// TIA Portal V16 export
// export: Created 2023-03-29T11:05:02.9769249Z, ExportSetting WithDefaults, DisplayName Totally Integrated Automation Portal, DisplayVersion V16 Update 6, DisplayName TIA Portal Version Control Interface, DisplayVersion V16 Update 2, DisplayName TIA Portal Openness, DisplayVersion V16 Update 6, DisplayName STEP 7 Professional, DisplayVersion V16 Update 6, DisplayName STEP 7 Safety, DisplayVersion V16, DisplayName WinCC Advanced, DisplayVersion V16 Update 6
DATA_BLOCK "dbtags_Sterowanie"   // DB1
{ S7_Optimized_Access := 'FALSE' }
VERSION : 0.1
// stored: AutoNumber false, DBAccessibleFromOPCUA true, IsOnlyStoredInLoadMemory false, IsWriteProtectedInAS false
   VAR RETAIN
      PID_Compact : Struct
         Setpoint : Real := 1.5;
         Input : Real;
         Input_PER : Int;
         Disturbance : Real;
         ManualEnable : Bool;
         ManualValue : Real;
         ErrorAck : Bool;
         Reset : Bool;
         ModeActivate : Bool;
         Mode : Int := 3;
         ScaledInput : Real;
         Output : Real;
         Output_PER : Int;
         Output_PWM : Bool;
         SetpointLimit_H : Bool;
         SetpointLimit_L : Bool;
         InputWarning_H : Bool;
         InputWarning_L : Bool;
         State : Int;
         Error : Bool;
         ErrorBits : DWord;
      END_STRUCT;
      Tuning : Struct
         Mode : Int := 1;
         Mode_visible : Bool;
         SUT_visible : Bool;
         TIR_visible : Bool;
         last_state : Int;
      END_STRUCT;
      HMI : Struct
         PhysicalUnit : String[5] := '1/min';
         Output_PWM_USInt : USInt;
         "position reached" : Bool;
         ManualMode_visible : Bool;
         Setpoint_limited : Bool;
         ErrorBits_Int : Int;
         ErrorAck_Int : Int;
         Warning_Int : Int;
         ErrorAck_Int_edge : Bool;   // pamięć zbocza reset PID po error
         ErrorAck : Bool;   // reset błędu PID
         Acknowledge_visible : Bool;
      END_STRUCT;
      Speed : Struct
         encoder : Real;
         rpm : Real;
      END_STRUCT;
      SetupControlPompownia : Struct
         SV : Real := 2.0;
         r_Pv_Norm_OUT_2 : Real := 10.0;   // Zakres górny wejścia In_PER_PID
         r_Pv_Norm_OUT_1 : Real := 0.0;   // Zakres dolny wejścia In_PER_PID
         r_Lmn_Hlm : Real := 100.0;   // Ograniczenie górne wartości procesowej [%] MV
         r_Lmn_Llm : Real := 0.0;   // Ograniczenie dolne wartości procesowej [%] MV
         r_Sp_Hlm : Real := 10.0;   // Ograniczenie H zakresu zadawania wartości ciśnienie SV
         r_Sp_Llm : Real := 0.0;   // Ograniczenie L zakresu zadawania wartości ciśnienia SV
         r_Pv_HWrn : Real;   // Ostrzeżenie wysoki dla PV
         r_Pv_LWrn : Real;   // Ostrzeżenie niski dla PV
         r_Pv_Hlm : Real := 16.0;   // Przetwornik Limit górny
         r_Pv_Llm : Real := 0.0;   // Przetwornik Limit dlolny
         Time_ONK1 : Int := 20;
         Time_ONK2 : Int := 60;
         Time_OFFK1 : Int := 15;
         Time_OFFK2 : Int := 5;
         TimeHz : Int := 10;
         NO4_Cureent : Real;   // Aktualna zawartość amoniaku
         CureentValue_O2_1 : Real;   // Przyrost ciśnienia 1
         CureentValue_O2_2 : Real;   // Przyrost ciścienia 2
         Data_sek1 : Int;   // Licznik sekund dla pomiaru nr1 funkcji Calculation_of_the_increment
         Data_sek2 : Int;   // Licznik sekund dla pomiaru nr2 funkcji Calculation_of_the_increment
         Static_1 : Word;
         Z11_Status : Word;   // Status napędu copia z SCADA
         Z12_Status : Word;   // Status napędu copia z SCADA
         Static_2 : Real;
         Switch_Aut_Rem_Pompy : Bool;   // Bit przełacznika trybu pracy pomp
         tagsdbSwitch_ModelSterowania : Word;   // Wybur model sterowania0- wyłączone, 1- Dosilanie, 2- Przetłączanie, 3- Automat, 4- Ręczne
         barMax_Manual_Hz : Real := 5.0;   // Instancja wartości zadawanej w trybie manual do regulatora PID gdy ciśnienie w rurociągu max
         CurrentMax_Manual_Hz : Real := 5.0;   // Instancja wartości zadawanej w trybie manual do regulatora PID gdy przeciążony falownik
         Statut_Motor : Byte;   // Byte stanu gotowości pomp
         Mem_Res_setCMD_MC_P1 : Bool;   // Znacznik 50 Hz podtrzymanie przełączenia na sieć
         Mem_Res_setCMD_MC_P2 : Bool;   // Znacznik 50 Hz podtrzymanie przełączenia na sieć
         Mem_Res_setCMD_MC_P3 : Bool;   // Znacznik 50 Hz podtrzymanie przełączenia na sieć
         Switch_In_Analog_Mudbas : Bool;   // Bit przełączeania pomiędzy sygnałem bar z wej analog / Modbus
         PV_HWrn_correction : Real;   // Wspóczninik służący wprowadzeniu korekty ostrzeżenia przekroczenia wartości zadanej ciśnienie
         PV_LWrn_correction : Real;   // Wspóczninik służący wprowadzeniu korekty ostrzeżenia zbyt niskia wartości ciśnieniea w stosunku do zadanej
         TimerSet_O2_Up : IEC_TIMER;   // Czas opóżninia podniesienia zadanej wartości ciśnienia
         TimerSet_O2_Down : IEC_TIMER;   // Czas opóżninia obniżenia zadanej wartości ciśnienia
         Pv_Llm_B8 : Real := -1.0;   // Limit dolny przetwornika ciśnienie B8
         Pv_Hlm_B8 : Real := 2.0;   // Limit górny przetwornika ciśnienia B8
         set_a : Int;
         set_b : Int := 0;
         Setpoint_Inverter_Pompy { ExternalAccessible := 'False'; ExternalVisible := 'False'; ExternalWritable := 'False'} : Real;   // Wartość zadana Hz odczytane z Modbus
         Frequency_inverter_Pompy { ExternalAccessible := 'False'; ExternalVisible := 'False'; ExternalWritable := 'False'} : Real;   // Aktualne Hz silniku odczytane z Modbus
         MotorCurrent_Inverter_Pompy { ExternalAccessible := 'False'; ExternalVisible := 'False'; ExternalWritable := 'False'} : Real;   // Prąd na silniku zasilanym z falownika odczytane z Modbus
         NormalCurrent_InverterPompy { ExternalAccessible := 'False'; ExternalVisible := 'False'; ExternalWritable := 'False'} : Real;   // Prąd nominalny falownika odczytane z Modbus
         MaxCurrent_Inverter_Pompy { ExternalAccessible := 'False'; ExternalVisible := 'False'; ExternalWritable := 'False'} : Real;   // Prad Max krótkotrwały odczytane z Modbus
         OverTemp_InverterPompy { ExternalAccessible := 'False'; ExternalVisible := 'False'; ExternalWritable := 'False'} : Word;
         OverVolta_InverterPompy { ExternalAccessible := 'False'; ExternalVisible := 'False'; ExternalWritable := 'False'} : Word;
         PIF_Reset : IEC_TIMER;   // impuls resetu regulatora PID 1
         mbAdresMPP04_Q1 : Word := 6;   // Adres modbus przepływomierz pompownia
         mbAdresPompy : Word := 26;   // Adres modbus falownik
         mbAdresMPP04_Q2 : Word;   // Adres modbus przepływomierz magistrala - w Stacji Zasuw
         mbAdres_IDslave : Word := 2;   // Adres modbus MT101
         SubPV_K1 : Real := 0.6;   // Wspólczynnik pomniejszenia wyliczanego ciśnienia napotrzeby wyłączenia dodatowej pompy
         SubPV_K2 : Real := 0.45;   // Wspólczynnik pomniejszenia wyliczanego ciśnieia napotrzeby wyłączenia dodatowej pompy
         Setpoint_Inverter_a { ExternalAccessible := 'False'; ExternalVisible := 'False'; ExternalWritable := 'False'} : Real;   // Wartość zadana Hz odczytane z Modbus
         Frequency_inverter_a { ExternalAccessible := 'False'; ExternalVisible := 'False'; ExternalWritable := 'False'} : Real;   // Aktualne Hz silniku odczytane z Modbus
         MotorCurrent_Inverter_a { ExternalAccessible := 'False'; ExternalVisible := 'False'; ExternalWritable := 'False'} : Real;   // Prąd na silniku zasilanym z falownika odczytane z Modbus
         NormalCurrent_Inverter_a { ExternalAccessible := 'False'; ExternalVisible := 'False'; ExternalWritable := 'False'} : Real;   // Prąd nominalny falownika odczytane z Modbus
         MaxCurrent_Inverter_a { ExternalAccessible := 'False'; ExternalVisible := 'False'; ExternalWritable := 'False'} : Real;   // Prad Max krótkotrwały odczytane z Modbus
         OverTemp_InverterPomp { ExternalAccessible := 'False'; ExternalVisible := 'False'; ExternalWritable := 'False'} : Word;
         OverVolta_InverterPomp { ExternalAccessible := 'False'; ExternalVisible := 'False'; ExternalWritable := 'False'} : Word;
         set_barDN500_B5 { ExternalAccessible := 'False'; ExternalVisible := 'False'; ExternalWritable := 'False'} : Real;   // Zadane ciśnienie dosilanie DN500 na czujniku B5
         set_barDN225_B6 { ExternalAccessible := 'False'; ExternalVisible := 'False'; ExternalWritable := 'False'} : Real;   // Zadane ciśnienie przetłacania DN225 na czujniku B6
         MotorCurrent_Inverter_b { ExternalAccessible := 'False'; ExternalVisible := 'False'; ExternalWritable := 'False'} : Real;   // Prąd na silniku zasilanym z falownika odczytane z Modbus
         NormalCurrent_Inverter_b { ExternalAccessible := 'False'; ExternalVisible := 'False'; ExternalWritable := 'False'} : Real;   // Prąd nominalny falownika odczytane z Modbus
         MaxCurrent_Inverter_b { ExternalAccessible := 'False'; ExternalVisible := 'False'; ExternalWritable := 'False'} : Real;   // Prad Max krótkotrwały odczytane z Modbus
         OverTemp_Inverter_b { ExternalAccessible := 'False'; ExternalVisible := 'False'; ExternalWritable := 'False'} : Word;
         OverVolta_Inverter_b { ExternalAccessible := 'False'; ExternalVisible := 'False'; ExternalWritable := 'False'} : Word;
         actOverCurrent_set : Real;   // Zakres ograniczenia prądowego.
         actOverCurrent_set_a : Real := 0.0;   // Zakres ograniczenia prądowego.
         actOverCurrent_set_b : Real := 0.0;   // Zakres ograniczenia prądowego.
         AnalogFrequency_inverter_a { ExternalAccessible := 'False'; ExternalVisible := 'False'; ExternalWritable := 'False'} : Real;   // Aktualne Hz silniku odczytane z Analog
         AnalogFrequency_inverter_b { ExternalAccessible := 'False'; ExternalVisible := 'False'; ExternalWritable := 'False'} : Real := 0.0;   // Aktualne Hz silniku odczytane z Analog
         MaxHour_InverterBlowerWork : Word := 43200;   // Maksymalny czas pracy pracy ciągłej na falowniku dla kompresorów 43200sek = 12h
         TimerSet_Hz_Up_a : IEC_TIMER;
         TimerSet_Hz_Down_a : IEC_TIMER;
         TimerSet_Hz_Up_b : IEC_TIMER;
         TimerSet_Hz_Down_b : IEC_TIMER;
         TimerGen_Hz_Up_a : IEC_TIMER;
         TimerGen_Hz_Down_a : IEC_TIMER;
         TimerGen_Hz_Up_b : IEC_TIMER;
         TimerGen_Hz_Down_b : IEC_TIMER;
         Mem_Res_setCMD_MC_P4 : Bool;   // Znacznik 50 Hz podtrzymanie przełączenia na sieć
         "MPP04_1Master.mode" : Byte := 0;
         "MPP04_2Master.mode" : Byte := 0;
         "Fal_2Master.mode_1" : Byte := 0;
         "Slave_2Master.mode_2" : Byte := 2;
      END_STRUCT;
      "Paramaetry _Zbiorniki" : Struct   // parametry sterowania
         set_poziom_napełniania : Real := 550.0;   // wartość zadana poziomu napełniania
         set_poziom_opróżniania : Real := 30.0;   // wartość zadana poziomu opróżniania
         set_bity_sterowania_napęami_1 : Word;   // bity sterowania napędami
         set_bity_sterowania_napęami_2 : Word;   // bity sterowania napędami
         set_bity_tryb_napędów_1 : Word;   // bity sterowania przełączaniem trybów pracy
         set_bity_tryb_napędów_2 : Word;   // bity sterowania przełączaniem trybów pracy
         rez_alarm_napędów : Word;   // bity kasowania alarmów napędów
         set_strategia_sterowania : Word;   // Sygnały sterowania strategią pompownia - 0= wyłaczone, 1=dosilanie, 2=przetłaczanie,3=automat, 4=ręczne
         set_sterowanie_cyklem : Word;   // Sygnały sterowania cyklem zbiorniki 0-wyłączone, 1=dobowy, 2=tygodniowy, 3=ręczne
         set_położenie_Z10 : Word;   // zadane położenie procentowe Z10
      END_STRUCT;
      Zbiorniki_Godziny : Struct   // godziny cykli pracy
         start_napełnianie : DTL := DTL#1970-01-01-23:55:00;
         Stop_napełnianie : DTL := DTL#1970-01-01-16:00:00;
         Start_przetłaczanie_1 : DTL := DTL#1970-01-01-18:00:00;
         Stop_przetłaczanie_1 : DTL := DTL#1970-01-01-23:55:00;
         Start_dosilanie_1 : DTL := DTL#1970-01-01-18:00:00;
         Stop_dosilanie_1 : DTL := DTL#1970-01-01-23:55:00;
      END_STRUCT;
   END_VAR
BEGIN
   SetupControlPompownia.PIF_Reset.PT := T#500ms;
   SetupControlPompownia.TimerSet_Hz_Up_a.PT := T#2M;
   SetupControlPompownia.TimerSet_Hz_Down_a.PT := T#2M;
   SetupControlPompownia.TimerSet_Hz_Up_b.PT := T#2M;
   SetupControlPompownia.TimerSet_Hz_Down_b.PT := T#2M;
   SetupControlPompownia.TimerGen_Hz_Up_a.PT := T#100ms;
   SetupControlPompownia.TimerGen_Hz_Down_a.PT := T#100ms;
   SetupControlPompownia.TimerGen_Hz_Up_b.PT := T#100ms;
   SetupControlPompownia.TimerGen_Hz_Down_b.PT := T#100ms;
END_DATA_BLOCK
